PROGRAM MAIN
VAR
END_VAR

PRG_DIAGNOSTIC();
PRG_GMD();

//MG
PRG_INJ();
PRG_PressureControl();
//PRG_VGP(); // Keep commented out, test VGP  through axis until positions are verfified

END_PROGRAM

(* stored: Version 1.1.0.1, ProductVersion 3.1.4022.12
   POU MAIN: Id {80634dbc-d649-47af-a183-d3f1342ca1c9}, SpecialFunc None *)
